FUNCTION_BLOCK F_TO_C_CONV2 (* Template for a Simple Function Block Type *)
  (* Standard: 61499-1 *)
  (* Version 1.0, 2018-12-03, badger *)
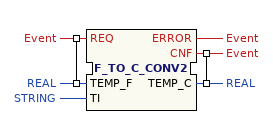
  EVENT_INPUT
    REQ WITH TEMP_F; (* Normal Execution Request *)
  END_EVENT
  EVENT_OUTPUT
    ERROR;
    CNF WITH TEMP_C; (* Execution Confirmation *)
  END_EVENT
  VAR_INPUT
    TEMP_F : REAL; (* Fahrenheit temperature to be converted *)
    TI : STRING;
  END_VAR
  VAR_OUTPUT
    TEMP_C : REAL; (* Converted temperature in celcius *)
  END_VAR
  ALGORITHM REQ IN ST: (* Normally executed algorithm *)
	ERROR() = FALSE;
	OUT() =  (IN() - 32) * 5 / 9;
	IF (OUT() < -273) {
		ERROR() = TRUE;
	}
  END_ALGORITHM
END_FUNCTION_BLOCK
